FUNCTION_BLOCK ASR_LAST_2 (* MERGE 2 ASR in 1 ASR (letztes Event gewinnt, reines Event-Fan-in - ASR traegt keine Nutzdaten, daher kein ECC noetig) *)
  (* Standard: 61499-2; Description: Copyright (c) 2026 Meisterschulen am Ostbahnhof This program and the accompanying materials are made available under the terms of the Eclipse Public License 2.0 which is available at https://www.eclipse.org/legal/epl-2.0/ SPDX-License-Identifier: EPL-2.0 *)
  (* Version 1.0, 2026-08-31, Franz Höpfinger, Meisterschulen am Ostbahnhof, pure event fan-in composite - both Sockets' events feed the same Plug event(s) directly; legal in 4diac since EventConnections (unlike DataConnections) allow multiple sources into one destination *)
  PACKAGE adapter::events::unidirectional;
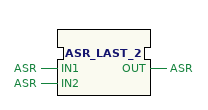
  SOCKETS
    IN1 : adapter::types::unidirectional::ASR;
    IN2 : adapter::types::unidirectional::ASR;
  END_SOCKETS
  PLUGS
    OUT : adapter::types::unidirectional::ASR;
  END_PLUGS
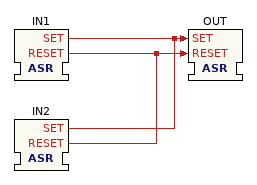
  EVENT_CONNECTIONS
    IN1.SET TO OUT.SET;
    IN2.SET TO OUT.SET;
    IN1.RESET TO OUT.RESET;
    IN2.RESET TO OUT.RESET;
  END_CONNECTIONS
END_FUNCTION_BLOCK
